// TIA Portal V17 export
// export: Created 2022-03-12T16:05:33.8479734Z, ExportSetting WithDefaults, DisplayName Totally Integrated Automation Portal, DisplayVersion V17, DisplayName TIA Portal Openness, DisplayVersion V17, DisplayName TIA Portal Version Control Interface, DisplayVersion V17, DisplayName STEP 7 Professional, DisplayVersion V17, DisplayName STEP 7 Safety, DisplayVersion V17, DisplayName WinCC Advanced / Unified PC, DisplayVersion V17
TYPE "CPG_typeProdCount(DINT)"
// stored: IsFailsafeCompliant false
   STRUCT
      ID : DInt;   // Product ID - This is the arbitrary (user defined) ID value of the consumed production material
      "Name" : String[24];   // Descriptive name - The name is used to literally describe the material ID, and its associated material
      Unit : String[5];   // Unit of measure - The unit tag is used to describe the names associated with a specific material used by the machine
      Count : DInt;   // Value - The count value is used as a variable for displaying information about the amount of consumed
      AccCount : DInt;   // Value - The accumulative count value is used as a variable for displaying information about the total amount of consumed production material
   END_STRUCT;
END_TYPE
